// TIA Portal V20 export
// export: Created 2026-07-22T09:47:30.5115567Z, ExportSetting WithDefaults, DisplayName Totally Integrated Automation Portal, DisplayVersion V20, DisplayName TIA Portal Openness, DisplayVersion V20, DisplayName TIA Portal Version Control Interface, DisplayVersion V20, DisplayName STEP 7 Professional, DisplayVersion V20, DisplayName STEP 7 Safety, DisplayVersion V20, DisplayName WinCC Basic/Comfort/Advanced, DisplayVersion V20, DisplayName WinCC Professional, DisplayVersion V20, DisplayName WinCC Unified, DisplayVersion V20
DATA_BLOCK "HMI_Interface_DB"   // DB7
{ S7_Optimized_Access := 'TRUE' }
VERSION : 0.1
// stored: AutoNumber true, IsOnlyStoredInLoadMemory false, IsRetainMemResEnabled false, IsWriteProtectedInAS false, MemoryReserve 100
   VAR
      SelectedValveIndex : Int;
      OpenCmd : Bool;
      CloseCmd : Bool;
      OpenFB : Bool;
      ClosedFB : Bool;
      Healthy : Bool;
      LocalMode : Bool;
   END_VAR
BEGIN
END_DATA_BLOCK
